{attribute 'GeneratedUsingTerminal: EL4112--0000'}
{attribute addProperty BoxType "EL4112--0000"}
{attribute addProperty Description "EL4112 2Ch. Ana. Output 0-20mA"}
{attribute addProperty Physics "KK"}
{attribute addProperty Id "Channel_1AT %Q*Channel_5F9B7EA62Channel_2AT %Q*Channel_5F9B7EA62WcStateAT %I*WcState_0B2B16F91InfoDataAT %I*InfoData_32EB74EA10"}
{attribute addProperty CRC "695255852"}
{attribute addProperty Size "15"}
TYPE EL4112_2970C32C EXTENDS EtcSlaveTerminalBase_947E5A46 :
STRUCT
	{attribute addProperty Name "Channel_1"}
	Channel_1 : Channel_5F9B7EA6;
	{attribute addProperty Name "Channel_2"}
	Channel_2 : Channel_5F9B7EA6;
	{attribute addProperty Name "WcState"}
	WcState : WcState_0B2B16F9;
	{attribute addProperty Name "InfoData"}
	InfoData : InfoData_32EB74EA;
END_STRUCT
END_TYPE

(* stored: Version 1.2.0.0, ProductVersion 3.1.4024.11
   DUT EL4112_2970C32C: Id {74498c9e-8307-4b38-8727-ede51dce79d1} *)
